FUNCTION_BLOCK FB_CrectCamUpDown_2	
VAR_INPUT
   	bCreatTable		                         :BOOL;	
	Reset                                        :BOOL;  
	iTable		                                :UINT;    
	 iTableSel		                             :UINT:=1;      //凸轮选择 
     bCamIn		                                 :BOOL;	
	

	fInitLength									:REAL;//耦合的初始高度
    fMoveLength                              :REAL;   //目标取或放料高度
    fSaveLength                               :REAL;    //升降安全高度

    fMasterKeyPos1                           :REAL:=208;   
    fMasterKeyPos2                           :REAL:=225;   
	fMasterKeyPos3                           :REAL:=256;   
    fMasterKeyPos4                           :REAL:=328;   
	fMasterKeyPos5                           :REAL:=328;   
	fSlaveVelo                                    :REAL:=0.32;   	
END_VAR

VAR_IN_OUT
	axisSlave		                            :axis_ref;  
	axisMaster		                            :axis_ref;  
END_VAR

VAR_OUTPUT
    bCreatTableDone                        :BOOL;
    bCreatTableError                        :BOOL;
	bError                         :BOOL;

END_VAR


VAR
	rtrigs		                                      :ARRAY[1..3]OF R_TRIG;
	ftrigs		                                      :ARRAY[1..3]OF F_TRIG;
    PositionData1			                  :ARRAY[1..7] OF MC_MotionFunctionPoint;	////
	fbCamtableselect:		               	MC_CamTableSelect;////
	Cam_table:				MC_CAM_REF;////
	bWriteCamData: BOOL;
    iCreatTableStep       :INT;
	
	rtTableChange:Tc2_Standard.R_TRIG;
   fbChangeCamModeSet	:	MC_SetCamOnlineChangeMode;
   fbModifyPoints		:ARRAY[1..4] OF	 MC_WriteMotionFunctionPoint;
   fbCamInSlave: BOOL;
   MA1: BOOL;
    bInSync: INT;
	
	
	
	iTableSelTemp: UINT;
END_VAR


rtrigs[1](CLK:=bCreatTable);  
ftrigs[1](CLK:=bCreatTable);  

CASE iCreatTableStep OF   
0:  
    IF  rtrigs[1].Q  AND NOT bCreatTableError  THEN
         fbCamtableselect.Execute:=FALSE;
         bCreatTableDone:=FALSE;
         bCreatTable:=FALSE;
         bWriteCamData:=TRUE;
         iCreatTableStep:=10;
    END_IF 

10: 
   IF NOT bWriteCamData THEN 
	  fbCamtableselect.Execute:=TRUE;   
	 iCreatTableStep:=20;	
  END_IF

20:		
	IF NOT  fbCamtableselect.Execute   THEN
        bCreatTableDone:=TRUE;
		iCreatTableStep:=0;	
    ELSIF  fbCamtableselect.Error        THEN
       bCreatTableError:=TRUE;
       iCreatTableStep:=999;	//创建凸轮失败
	END_IF		
END_CASE

(**********故障***********)
	IF  Reset  AND bCreatTableError  THEN  
	   bCreatTableError:=FALSE;
	   iCreatTableStep:=0;
	END_IF


ModifyCam();

ACTION ModifyCam:

fbCamtableselect(   
	Execute:=                        fbCamtableselect.Execute ,
	Periodic:=                        FALSE ,
	MasterAbsolute:=             FALSE,
	SlaveAbsolute:=                FALSE ,
	CamTableID:=                  iTable,
	Master:=                         axisMaster ,
	Slave:=                            axisSlave ,
	CamTable:=                     Cam_table , );

IF fbCamtableselect.Done THEN
    fbCamtableselect.Execute:=FALSE;
END_IF



IF bWriteCamData  THEN
 
	  Cam_table.ArraySize:=SIZEOF(PositionData1); 
	  Cam_table.NoOfColumns:=1;
	  Cam_table.NoOfRows:=7;
	  Cam_table.pArray:=ADR(PositionData1);
	  Cam_table.TableType:=MC_TABLETYPE_MOTIONFUNCTION;
  
      //MOTIONFUNCTYPE_BESCHLTRAPEZ     MOTIONFUNCTYPE_POLYNOM7_MM    MOTIONFUNCTYPE_BESCHLTRAPEZ   MOTIONFUNCTYPE_POLYNOM1

	  PositionData1[1].	PointIndex	:=	        1;
	  PositionData1[1].	FunctionType	:=		MOTIONFUNCTYPE_POLYNOM5_MM;//MOTIONFUNCTYPE_BESCHLTRAPEZ     MOTIONFUNCTYPE_POLYNOM7_MM    MOTIONFUNCTYPE_BESCHLTRAPEZ
	  PositionData1[1].	PointType	:=	        MOTIONPOINTTYPE_MOTION;
	  PositionData1[1].	RelIndexNextPoint	:=  1;
	  PositionData1[1].	MasterPos	:=	        0;
	  PositionData1[1].	SlavePos	:=	        0;		//fMoveLength
	  PositionData1[1].	SlaveVelo	:=	        0;
	  
	  PositionData1[2].	PointIndex	:=	        2;
	  PositionData1[2].	FunctionType	:=		MOTIONFUNCTYPE_POLYNOM5_MM;
	  PositionData1[2].	PointType	:=	        MOTIONPOINTTYPE_MOTION;
	  PositionData1[2].	RelIndexNextPoint	:=  1;
	  PositionData1[2].	MasterPos	:=	        fMasterKeyPos1;//fMasterKeyPos
	  PositionData1[2].	SlavePos	:=	        fSaveLength ;	
	  PositionData1[2].	SlaveVelo	:=	        0;//(fInitLength-fSaveLength)/fMasterKeyPos1	;
	  
	  PositionData1[3].	PointIndex	:=	        3;
	  PositionData1[3].	FunctionType	:=		MOTIONFUNCTYPE_POLYNOM5_MM;
	  PositionData1[3].	PointType	:=	        MOTIONPOINTTYPE_MOTION;
	  PositionData1[3].	RelIndexNextPoint	:=  1;
	  PositionData1[3].	MasterPos	:=	        fMasterKeyPos2;//fMasterKeyPos
	  PositionData1[3].	SlavePos	:=	        fMoveLength-4;	
	  PositionData1[3].	SlaveVelo	:=	        fSlaveVelo;//(fInitLength-fSaveLength)/fMasterKeyPos1	;  
	  
	  PositionData1[4].	PointIndex	:=	        4;
	  PositionData1[4].	FunctionType	:=		MOTIONFUNCTYPE_POLYNOM1;
	  PositionData1[4].	PointType	:=	        MOTIONPOINTTYPE_MOTION;
	  PositionData1[4].	RelIndexNextPoint	:=  1;
	  PositionData1[4].	MasterPos	:=	        fMasterKeyPos3;
	  PositionData1[4].	SlavePos	:=	        fMoveLength;	
	  PositionData1[4].	SlaveVelo	:=	        0	;

	  PositionData1[5].	PointIndex	:=	        5;
	  PositionData1[5].	FunctionType	:=		MOTIONFUNCTYPE_POLYNOM5_MM;
	  PositionData1[5].	PointType	:=	        MOTIONPOINTTYPE_MOTION;
	  PositionData1[5].	RelIndexNextPoint	:=  1;
	  PositionData1[5].	MasterPos	:=	        fMasterKeyPos4;//fMasterKeyPos
	  PositionData1[5].	SlavePos	:=	        fMoveLength;	
	  PositionData1[5].	SlaveVelo	:=	       0	;

	  PositionData1[6].	PointIndex	:=	        6;
	  PositionData1[6].	FunctionType	:=		MOTIONFUNCTYPE_POLYNOM5_MM;
	  PositionData1[6].	PointType	:=	        MOTIONPOINTTYPE_MOTION;
	  PositionData1[6].	RelIndexNextPoint	:=  1;
	  PositionData1[6].	MasterPos	:=	        fMasterKeyPos5;
	  PositionData1[6].	SlavePos	:=	        0;	
	  PositionData1[6].	SlaveVelo	:=	       0	;

	  PositionData1[7].	PointIndex	:=	        7;
	  PositionData1[7].	FunctionType	:=		MOTIONFUNCTYPE_POLYNOM5_MM;
	  PositionData1[7].	PointType	:=	        MOTIONPOINTTYPE_MOTION;
	  PositionData1[7].	RelIndexNextPoint	:=  0;
	  PositionData1[7].	MasterPos	:=	        360;
	  PositionData1[7].	SlavePos	:=	        0;	
	  PositionData1[7].	SlaveVelo	:=	       0	;

     bWriteCamData:=FALSE;
END_IF



(*
IF bWriteCamData  THEN
 
	  Cam_table.ArraySize:=SIZEOF(PositionData1); 
	  Cam_table.NoOfColumns:=1;
	  Cam_table.NoOfRows:=7;
	  Cam_table.pArray:=ADR(PositionData1);
	  Cam_table.TableType:=MC_TABLETYPE_MOTIONFUNCTION;
  
      //MOTIONFUNCTYPE_BESCHLTRAPEZ     MOTIONFUNCTYPE_POLYNOM7_MM    MOTIONFUNCTYPE_BESCHLTRAPEZ   MOTIONFUNCTYPE_POLYNOM1

	  PositionData1[1].	PointIndex	:=	        1;
	  PositionData1[1].	FunctionType	:=		MOTIONFUNCTYPE_POLYNOM5_MM;//MOTIONFUNCTYPE_BESCHLTRAPEZ     MOTIONFUNCTYPE_POLYNOM7_MM    MOTIONFUNCTYPE_BESCHLTRAPEZ
	  PositionData1[1].	PointType	:=	        MOTIONPOINTTYPE_MOTION;
	  PositionData1[1].	RelIndexNextPoint	:=  1;
	  PositionData1[1].	MasterPos	:=	        0;
	  PositionData1[1].	SlavePos	:=	        0;		//fMoveLength
	  PositionData1[1].	SlaveVelo	:=	        0;
	  
	  PositionData1[2].	PointIndex	:=	        2;
	  PositionData1[2].	FunctionType	:=		MOTIONFUNCTYPE_POLYNOM5_MM;
	  PositionData1[2].	PointType	:=	        MOTIONPOINTTYPE_MOTION;
	  PositionData1[2].	RelIndexNextPoint	:=  1;
	  PositionData1[2].	MasterPos	:=	        fMasterKeyPos1;//fMasterKeyPos
	  PositionData1[2].	SlavePos	:=	        fSaveLength - fInitLength;	
	  PositionData1[2].	SlaveVelo	:=	        0;//(fInitLength-fSaveLength)/fMasterKeyPos1	;

	  PositionData1[3].	PointIndex	:=	        3;
	  PositionData1[3].	FunctionType	:=		MOTIONFUNCTYPE_POLYNOM5_MM;
	  PositionData1[3].	PointType	:=	        MOTIONPOINTTYPE_MOTION;
	  PositionData1[3].	RelIndexNextPoint	:=  1;
	  PositionData1[3].	MasterPos	:=	        fMasterKeyPos2;//fMasterKeyPos
	  PositionData1[3].	SlavePos	:=	        0;	
	  PositionData1[3].	SlaveVelo	:=	        0;//(fInitLength-fSaveLength)/fMasterKeyPos1	;
	  
	  PositionData1[4].	PointIndex	:=	        4;
	  PositionData1[4].	FunctionType	:=		MOTIONFUNCTYPE_POLYNOM5_MM;
	  PositionData1[4].	PointType	:=	        MOTIONPOINTTYPE_MOTION;
	  PositionData1[4].	RelIndexNextPoint	:=  1;
	  PositionData1[4].	MasterPos	:=	        fMasterKeyPos3;
	  PositionData1[4].	SlavePos	:=	        fMoveLength-fInitLength-4;	
	  PositionData1[4].	SlaveVelo	:=	        4*0.7/(fMasterKeyPos4-fMasterKeyPos3)	;

	  PositionData1[5].	PointIndex	:=	        5;
	  PositionData1[5].	FunctionType	:=		MOTIONFUNCTYPE_POLYNOM5_MM;
	  PositionData1[5].	PointType	:=	        MOTIONPOINTTYPE_MOTION;
	  PositionData1[5].	RelIndexNextPoint	:=  1;
	  PositionData1[5].	MasterPos	:=	        fMasterKeyPos4;
	  PositionData1[5].	SlavePos	:=	        fMoveLength-fInitLength;	
	  PositionData1[5].	SlaveVelo	:=	        0	;	  
	  
	  PositionData1[6].	PointIndex	:=	        6;
	  PositionData1[6].	FunctionType	:=		MOTIONFUNCTYPE_POLYNOM5_MM;
	  PositionData1[6].	PointType	:=	        MOTIONPOINTTYPE_MOTION;
	  PositionData1[6].	RelIndexNextPoint	:=  1;
	  PositionData1[6].	MasterPos	:=	        fMasterKeyPos5;//fMasterKeyPos
	  PositionData1[6].	SlavePos	:=	        fMoveLength-fInitLength;	
	  PositionData1[6].	SlaveVelo	:=	       0	;

	  PositionData1[7].	PointIndex	:=	        7;
	  PositionData1[7].	FunctionType	:=		MOTIONFUNCTYPE_POLYNOM5_MM;
	  PositionData1[7].	PointType	:=	        MOTIONPOINTTYPE_MOTION;
	  PositionData1[7].	RelIndexNextPoint	:=  0;
	  PositionData1[7].	MasterPos	:=	        360;
	  PositionData1[7].	SlavePos	:=	        0;	
	  PositionData1[7].	SlaveVelo	:=	       0	;


     bWriteCamData:=FALSE;
END_IF

*)



fbChangeCamModeSet(
	Execute:=                              fbCamtableselect.Done OR MA1 ,
	ActivationMode:=                  MC_CAMACTIVATION_NEXTCYCLE ,				
	ActivationPosition:=               0.0 ,
	MasterScalingMode:=           MC_CAMSCALING_AUTOOFFSET ,
	SlaveScalingMode:=              MC_CAMSCALING_AUTOOFFSET ,
	CamTableID:=iTable,
	Done=>                                ,
	Busy=>                                  ,
	Error=>                                ,
	ErrorID=>                            );

	fbChangeCamModeSet.Done;
	fbChangeCamModeSet.Busy;
	fbChangeCamModeSet.Error;
	fbChangeCamModeSet.ErrorID;
	
(*	
rtTableChange(CLK:=axisMaster.Status.Moving AND axisSlave.Status.Coupled AND bInSync AND 
                              axisMaster.NcToPlc.ModuloActPos>350 AND axisMaster.NcToPlc.ModuloActPos<359  OR rtrigs[2].Q AND axisMaster.Status.NotMoving , Q=> );  
*)						  
							  
rtrigs[2](CLK:=bCamIn);  
//rtrigs[3](CLK:=bCreatTable);  

rtTableChange(CLK:=  rtrigs[2].Q  AND iTableSel <>iTableSelTemp , Q=> );  
	
IF   rtTableChange.Q THEN
                   
    IF  iTableSel=1 THEN   
	  PositionData1[4].	PointIndex	:=	        4;
	  PositionData1[4].	FunctionType	:=		MOTIONFUNCTYPE_POLYNOM1;
	  PositionData1[4].	PointType	:=	        MOTIONPOINTTYPE_MOTION;
	  PositionData1[4].	RelIndexNextPoint	:=  1;
	  PositionData1[4].	MasterPos	:=	        fMasterKeyPos3;
	  PositionData1[4].	SlavePos	:=	        fMoveLength;	
	  PositionData1[4].	SlaveVelo	:=	        0	;

	  PositionData1[5].	PointIndex	:=	        5;
	  PositionData1[5].	FunctionType	:=		MOTIONFUNCTYPE_POLYNOM5_MM;
	  PositionData1[5].	PointType	:=	        MOTIONPOINTTYPE_MOTION;
	  PositionData1[5].	RelIndexNextPoint	:=  1;
	  PositionData1[5].	MasterPos	:=	        fMasterKeyPos4;//fMasterKeyPos
	  PositionData1[5].	SlavePos	:=	        fMoveLength;	
	  PositionData1[5].	SlaveVelo	:=	       0	;

   END_IF

    IF  iTableSel=2 THEN 
		
	  PositionData1[4].	PointIndex	:=	        4;
	  PositionData1[4].	FunctionType	:=		MOTIONFUNCTYPE_POLYNOM1;
	  PositionData1[4].	PointType	:=	        MOTIONPOINTTYPE_MOTION;
	  PositionData1[4].	RelIndexNextPoint	:=  1;
	  PositionData1[4].	MasterPos	:=	        fMasterKeyPos3;
	  PositionData1[4].	SlavePos	:=	        fMoveLength-2;	
	  PositionData1[4].	SlaveVelo	:=	        0	;

	  PositionData1[5].	PointIndex	:=	        5;
	  PositionData1[5].	FunctionType	:=		MOTIONFUNCTYPE_POLYNOM5_MM;
	  PositionData1[5].	PointType	:=	        MOTIONPOINTTYPE_MOTION;
	  PositionData1[5].	RelIndexNextPoint	:=  1;
	  PositionData1[5].	MasterPos	:=	        fMasterKeyPos4;//fMasterKeyPos
	  PositionData1[5].	SlavePos	:=	        fMoveLength-2;	
	  PositionData1[5].	SlaveVelo	:=	       0	;	
	
   END_IF
    iTableSelTemp:=iTableSel;     
END_IF

fbModifyPoints[1]( 
	Execute:=rtTableChange.Q , 
	CamTableID:=iTable,
	PointID:=5 ,
	Point:=PositionData1[5] ,
	Done=> ,
	Busy=> ,
	Error=> ,
	ErrorID=> );

fbModifyPoints[2]( 
	Execute:=rtTableChange.Q , 
	CamTableID:=iTable,
	PointID:=6 ,
	Point:=PositionData1[6] ,
	Done=> ,
	Busy=> ,
	Error=> ,
	ErrorID=> );
(*
fbModifyPoints[3]( 
	Execute:=rtTableChange.Q , 
	CamTableID:=iTable,
	PointID:=3 ,
	Point:=PositionData[3] ,
	Done=> ,
	Busy=> ,
	Error=> ,
	ErrorID=> );

*)
END_ACTION

END_FUNCTION_BLOCK

(* stored: Version 1.1.0.1, ProductVersion 3.1.4024.12
   POU FB_CrectCamUpDown_2: Id {7911671e-9951-4a13-b7ad-7c9b6fd2eab5}, SpecialFunc None
   Action ModifyCam: Id {6b623ea7-378d-44a4-9b7b-b13deebe58e7} *)
